FUNCTION_BLOCK FB_CRYO_LN2_PRECOOL EXTENDS FB_CRYO_GEN_CTRL_BASE
VAR_INPUT
	in_lrTempK:				LREAL;			// Temperature input value [K]
	in_bTempValid:			BOOL := TRUE;	// Temperature Valid flag
	// Two parameters for decision making
	in_lrTempValveOpen:		LREAL := 91.27;		// Open  valve if temperature above this value [K]
	in_lrTempValveClose:	LREAL := 79.148;	// Close valve if temperature below this value [K]
END_VAR
VAR_OUTPUT
END_VAR
VAR
	// Status structure
	{attribute 'OPC.UA.DA' := '1'}
	stat:				T_CRYO_GEN_CTRL_STATUS_BASE;
	
	// LN2 valve
	valve:				FB_CRYO_VALVE_CTRL;
	bEnable_valve:		BOOL := FALSE;	// Valve open when bEnable_valve = TRUE
		

END_VAR

SUPER^();

METHOD M_ActionOffExecute
VAR_INPUT
END_VAR
//
// In this method the Enable flag of the valve is set to FALSE,
// meaning close the valve.
// 
// In the corresponding Activity M_ActivitySwitchingOff(), 
// the completion of the CLOSE/OFF command will be checked.
//
timer(IN:=FALSE);	// Reset Timer - mandatory!

// Close the valve
bEnable_valve	:= FALSE;
END_METHOD

METHOD M_ActionOnExecute
VAR_INPUT
END_VAR
//
// In this method the Enable flag of the valve is set to TRUE,
// meaning open the valve.
// 
// In the corresponding Activity M_ActivitySwitchingOn(), 
// the completion of the OPEN/ON command will be checked.
//
timer(IN:=FALSE);	// Reset Timer - mandatory!

// Close the valve
bEnable_valve	:= TRUE;
END_METHOD

METHOD M_ActivitySwitchingOff : BOOL
VAR_INPUT
END_VAR
//
// Wait for the valve to CLOSE/OFF.
// The valve state is available in its status structure.
// When complete, the method shall return TRUE, otherwise FALSE.


//
// Execute the timer - mandatory.
// Timer expiry is checked in M_ProcessEvents().
//
timer(IN:=TRUE, PT:=UDINT_TO_TIME(in_nTimeout));
	
// If valve is closed, return TRUE, otherwise FALSE.
IF valve.stat.bActOFF THEN
	M_ActivitySwitchingOff := TRUE;
ELSE
	M_ActivitySwitchingOff := FALSE;
END_IF
END_METHOD

METHOD M_ActivitySwitchingOn : BOOL
VAR_INPUT
END_VAR
//
// Wait for the valve to OPEN/ON.
// The valve state is available in its status structure.
// When complete, the method shall return TRUE, otherwise FALSE.


//
// Execute the timer - mandatory.
// Timer expiry is checked in M_ProcessEvents().
//
timer(IN:=TRUE, PT:=UDINT_TO_TIME(in_nTimeout));
	
// If valve is open, return TRUE, otherwise FALSE.
IF valve.stat.bActON THEN
	M_ActivitySwitchingOn := TRUE;
ELSE
	M_ActivitySwitchingOn := FALSE;
END_IF
END_METHOD

METHOD M_Configure
VAR_INPUT
END_VAR
// Configure the system and set the bConfigured flag to TRUE.

(*
	TODO USER: 
	- Set references to extended structures. e.g.
	     statRef REF=stat;
	- Configure the system.
*)

//	MUST be the very first line!!!
statRef REF=stat;

// The system has been configured
bConfigured := TRUE;
END_METHOD

METHOD M_ControlLoop : BOOL
VAR_INPUT
END_VAR
//
// This method implements the logic for controlling the LN2 valve.
// 
// The return value indicates if the valve should be OPEN/TRUE or CLOSED/FALSE
//
	
CASE statRef.nState OF
	E_CRYO_BIN_CTRL_STATE.ACTIVE_SWITCHING_ON,
	E_CRYO_BIN_CTRL_STATE.ACTIVE_ON:
		IF in_bTempValid AND in_lrTempK < in_lrTempValveClose THEN
			// Temperature too low.
			// Close the valve to stop cooling.
			M_ControlLoop	:= FALSE;
		ELSE
			// Keep the valve open
			M_ControlLoop	:= TRUE;
		END_IF

	E_CRYO_BIN_CTRL_STATE.ACTIVE_SWITCHING_OFF,
	E_CRYO_BIN_CTRL_STATE.ACTIVE_OFF:
		IF in_bTempValid AND in_lrTempK > in_lrTempValveOpen THEN
			// Temperature too high.
			// Open the valve to start cooling.
			M_ControlLoop	:= TRUE;
		ELSE
			// Keep the valve closed
			M_ControlLoop	:= FALSE;
		END_IF
ELSE
	// Keep the valve closed
	M_ControlLoop	:= FALSE;
END_CASE
END_METHOD

METHOD M_ExecuteActuators
VAR_INPUT
END_VAR
(*
	TODO USER: Execute all actuators, e.g. valve, heater, etc.
*)

valve(	in_nTimeout	:= 3000, 
		in_bEnable	:= bEnable_valve);
END_METHOD

METHOD M_IsError : BOOL
VAR_INPUT
END_VAR
//
// Check all possible failure conditions.
//
// This includes:
// - Configuration,
// - Validity of temperature reading,
// - Valve failure.
// 
// Return TRUE in case of errors.
// Set error description as well.
//
IF in_lrTempValveClose >= in_lrTempValveOpen THEN
	// The temperatue at which valve opens must be
	// higher than the one at which it closes.
	M_IsError	:= TRUE;
	stat.sError	:= 'ERROR: Wrong temperature limits!';
ELSIF NOT in_bTempValid	THEN
	// Temperature reading invalid.
	M_IsError	:= TRUE;
	stat.sError	:= 'ERROR: Reference temperature invalid!';
ELSIF valve.stat.bError 	THEN
	// Valve has failed.
	M_IsError	:= TRUE;
	stat.sError	:= 'ERROR: Valve failure!';
ELSE
	M_IsError	:= FALSE;
END_IF
END_METHOD

METHOD M_SetStatus
VAR_INPUT
END_VAR
// Execute M_SetStatus() of the base FB
SUPER^.M_SetStatus();


// Correct for LN2 specific labels

CASE statRef.nState OF
	
	E_CRYO_BIN_CTRL_STATE.ACTIVE_OFF:
	statRef.sState	:= 'ACTIVE_VALVE_CLOSED';
	
	E_CRYO_BIN_CTRL_STATE.ACTIVE_ON:
	statRef.sState	:= 'ACTIVE_VALVE_OPEN';
	
	E_CRYO_BIN_CTRL_STATE.ACTIVE_SWITCHING_ON:
	statRef.sState	:= 'OPENING VALVE...';
	
	E_CRYO_BIN_CTRL_STATE.ACTIVE_SWITCHING_OFF:
	statRef.sState	:= 'CLOSING VALVE...';
	
END_CASE
END_METHOD

END_FUNCTION_BLOCK

(* stored: Version 1.1.0.1, ProductVersion 3.1.4024.10
   POU FB_CRYO_LN2_PRECOOL: Id {01dbaf30-d219-4feb-bb44-39afda4b5c99}, SpecialFunc None
   Method M_ActionOffExecute: Id {914ec106-2ab3-47b6-8a78-a2c068ffcecc}
   Method M_ActionOnExecute: Id {c769b257-2ad7-4e3d-80ac-bd10fea18e00}
   Method M_ActivitySwitchingOff: Id {2541c467-5996-46ec-887b-4f36c70f21c2}
   Method M_ActivitySwitchingOn: Id {19c071f3-4450-4753-974a-78ee88d9e3d8}
   Method M_Configure: Id {f21ce1e8-203f-46f2-9062-ca50ece5da47}
   Method M_ControlLoop: Id {d2f77303-de70-4f2d-a948-f128b596ac02}
   Method M_ExecuteActuators: Id {9abf21cc-1b1d-432a-883c-7267a479b019}
   Method M_IsError: Id {5df1fcd2-ca20-405b-9600-d73bbdf7b059}
   Method M_SetStatus: Id {012a76b0-ddac-4b60-acc4-399fdb37cac5} *)
